// TIA Portal V17 export
// export: Created 2022-07-20T06:59:46.8680276Z, ExportSetting WithDefaults, DisplayName Totally Integrated Automation Portal, DisplayVersion V17, DisplayName TIA Portal Openness, DisplayVersion V17, DisplayName TIA Portal Version Control Interface, DisplayVersion V17, DisplayName SINAMICS Startdrive Advanced, DisplayVersion V17, DisplayName SINAMICS Startdrive G130, G150, S120, S150, SINAMICS MV, S210, DisplayVersion V17, DisplayName SINAMICS Startdrive G110M, G120, G120C, G120D, G120P, G115D, DisplayVersion V17, DisplayName STEP 7 Professional, DisplayVersion V17, DisplayName STEP 7 Safety, DisplayVersion V17, DisplayName WinCC Advanced, DisplayVersion V17
FUNCTION_BLOCK "FB10100_ModbusRtuManager"   // FB10100, LAD
TITLE = FB10100_ModbusRtuManager
{ S7_Optimized_Access := 'FALSE' }
AUTHOR : Jonathan
FAMILY : 1010x_MODBUS
VERSION : 1.0
// Release note : 
// 1.0 - Feature developped
// 
// Todo : 
// Générer une erreur si la communication reste en busy trop longtemps
// stored: AutoNumber false, IsIECCheckEnabled false, SetENOAutomatically false, UDAEnableTagReadback false
   VAR_INPUT
      InitialCall : Bool;
      ModbusPort : HW_ANY;
      ModbusBaudRate : UDInt;
      ModbusParity : UInt;
      StartCommunication : Bool;
      Reset : Bool;
      Max_ModbusSlaves : Int := 1;
   END_VAR
   VAR_OUTPUT
      Init_Done : Bool;
      Init_Error : Bool;
      Init_Status : Word;
      Comm_Done : Bool;
      Comm_Busy : Bool;
      Comm_Error : Bool;
      Comm_Status : Word;
   END_VAR
   VAR_IN_OUT
      CurrentSlaveNumber : Int;
      SlavesParameters : Array[1.."MAX_MODBUS_SLAVES"] of "stModbusRtuSlaveParameters";
      SlavesRequests : Array[1.."MAX_MODBUS_SLAVES"] of "stModbusRtuSlaveRequests";
      SlavesStates : Array[1.."MAX_MODBUS_SLAVES"] of "stModbusRtuSlaveStates";
   END_VAR
   VAR
      Modbus_Master_DB { ExternalAccessible := 'False'; ExternalVisible := 'False'; ExternalWritable := 'False'; S7_SetPoint := 'True'} : Modbus_Master;
      Modbus_Comm_Load_DB { S7_SetPoint := 'True'} : Modbus_Comm_Load;
   END_VAR
   VAR DB_SPECIFIC
      InitalisationDoneStored : Bool;
      LocalProcessStep : USInt;
      LocalCommRequest : Bool;
      LocalMode : USInt;
      LocalSlaveDataTemp { ExternalAccessible := 'False'; ExternalVisible := 'False'; ExternalWritable := 'False'; S7_SetPoint := 'True'} : "stModbusRtuDataPtr";
      LocalSlaveAdress : UInt;
      LocalSlaveDataAdress : UInt;
      Data_modbus_Dint { ExternalAccessible := 'False'; ExternalVisible := 'False'; ExternalWritable := 'False'} : DInt;
      Modbus_value_Number { ExternalAccessible := 'False'; ExternalVisible := 'False'; ExternalWritable := 'False'} : DInt;
      LocalSlaveDataLength : UInt;
      Data_modbus_Int : Int;
      TON_TimeOutNotDone { S7_SetPoint := 'True'} : TON_TIME;
      LocalSlaveCurrentNumber : Int;
   END_VAR
   VAR_TEMP
      LowWeight : Int;
      LowWeight_1 : Real;
      Highweight : Real;
   END_VAR
   // Modbus_Comm_Load_DB.STOP_BITS := 2;
BEGIN

REGION Network 1: Initilisation of the mode (4 = Half Duplex) / Put 4 value for Half Duplex mode
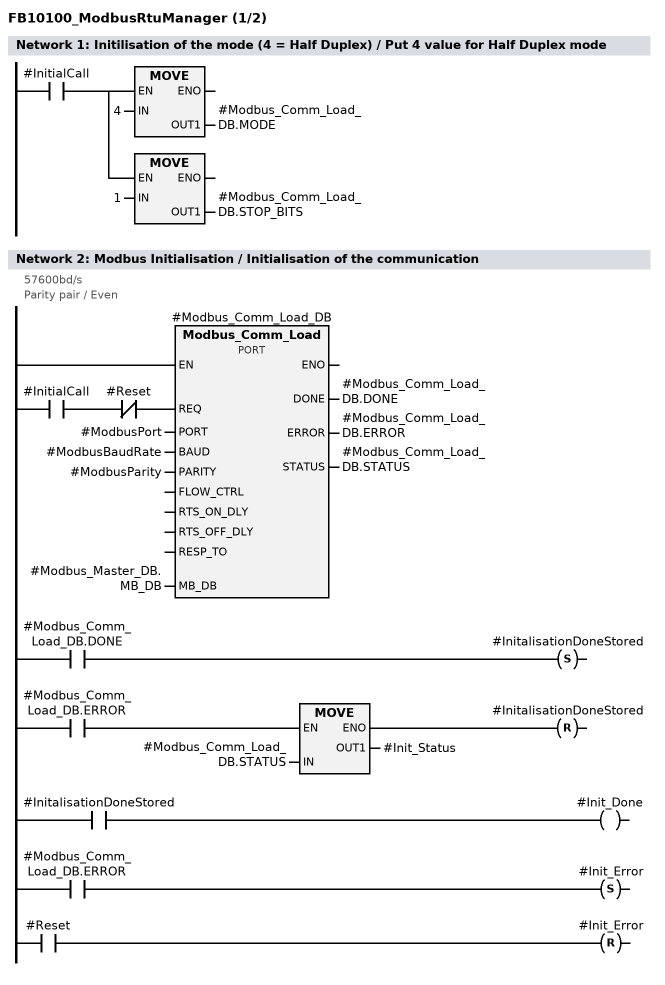
   RUNG wire#powerrail
      Contact( #InitialCall )
      wire#w1
      { S7_GenerateENO := "TRUE" } Move(in := 4, out1 => #Modbus_Comm_Load_DB.MODE)
   END_RUNG
   RUNG wire#w1
      { S7_GenerateENO := "TRUE" } Move(in := 1, out1 => #Modbus_Comm_Load_DB.STOP_BITS)
   END_RUNG
   // the same network as SCL:
   IF #InitialCall THEN
       #Modbus_Comm_Load_DB.MODE := 4;
       #Modbus_Comm_Load_DB.STOP_BITS := 1;
   END_IF;
END_REGION

REGION Network 2: Modbus Initialisation / Initialisation of the communication
   // 57600bd/s
   // Parity pair / Even
   RUNG wire#powerrail
      { S7_Templates := "[card := 0, port_type := PORT, word_type := UInt, dint_type := UDInt, mbbase_type := P2P_MB_BASE]" } #Modbus_Comm_Load_DB.Modbus_Comm_Load(REQ := wire#w1, PORT := #ModbusPort, BAUD := #ModbusBaudRate, PARITY := #ModbusParity, FLOW_CTRL :=, RTS_ON_DLY :=, RTS_OFF_DLY :=, RESP_TO :=, MB_DB := #Modbus_Master_DB.MB_DB, DONE => #Modbus_Comm_Load_DB.DONE, ERROR => #Modbus_Comm_Load_DB.ERROR, STATUS => #Modbus_Comm_Load_DB.STATUS)
   END_RUNG
   RUNG wire#powerrail
      Contact( #InitialCall )
      I_Contact( #Reset )
   END_RUNG wire#w1
   RUNG wire#powerrail
      Contact( #Modbus_Comm_Load_DB.DONE )
      S_Coil( #InitalisationDoneStored )
   END_RUNG
   RUNG wire#powerrail
      Contact( #Modbus_Comm_Load_DB.ERROR )
      { S7_GenerateENO := "TRUE" } Move(in := #Modbus_Comm_Load_DB.STATUS, out1 => #Init_Status)
      R_Coil( #InitalisationDoneStored )
   END_RUNG
   RUNG wire#powerrail
      Contact( #InitalisationDoneStored )
      Coil( #Init_Done )
   END_RUNG
   RUNG wire#powerrail
      Contact( #Modbus_Comm_Load_DB.ERROR )
      S_Coil( #Init_Error )
   END_RUNG
   RUNG wire#powerrail
      Contact( #Reset )
      R_Coil( #Init_Error )
   END_RUNG
   // the same network as SCL:
   // ENO of a box is taken as its EN; it also drops when the box reports an error
   #Modbus_Comm_Load_DB(REQ := #InitialCall AND NOT #Reset,   // Modbus_Comm_Load
                        PORT := #ModbusPort,
                        BAUD := #ModbusBaudRate,
                        PARITY := #ModbusParity,
                        MB_DB := #Modbus_Master_DB.MB_DB,
                        DONE => #Modbus_Comm_Load_DB.DONE,
                        ERROR => #Modbus_Comm_Load_DB.ERROR,
                        STATUS => #Modbus_Comm_Load_DB.STATUS);
   IF #Modbus_Comm_Load_DB.DONE THEN #InitalisationDoneStored := TRUE; END_IF;
   IF #Modbus_Comm_Load_DB.ERROR THEN
       #Init_Status := #Modbus_Comm_Load_DB.STATUS;
       #InitalisationDoneStored := FALSE;
   END_IF;
   #Init_Done := #InitalisationDoneStored;
   IF #Modbus_Comm_Load_DB.ERROR THEN #Init_Error := TRUE; END_IF;
   IF #Reset THEN #Init_Error := FALSE; END_IF;
END_REGION

REGION Network 3: Modbus Master Call / Master Exchange block
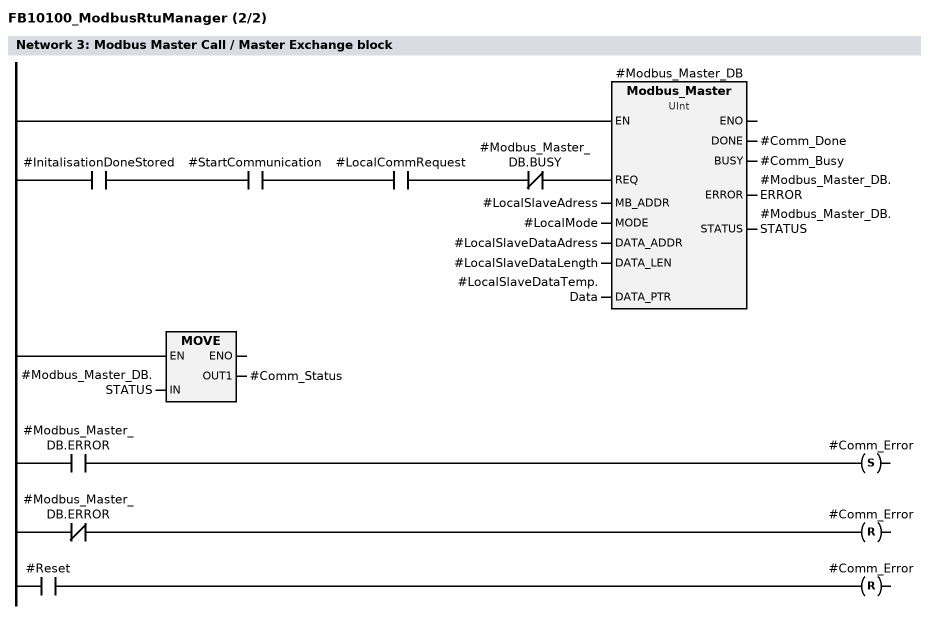
   RUNG wire#powerrail
      { S7_Templates := "[card := 0, word_type := UInt, dword_type := UDInt, byte_type := USInt, any_type := Variant]" } #Modbus_Master_DB.Modbus_Master(REQ := wire#w1, MB_ADDR := #LocalSlaveAdress, MODE := #LocalMode, DATA_ADDR := #LocalSlaveDataAdress, DATA_LEN := #LocalSlaveDataLength, DATA_PTR := #LocalSlaveDataTemp.Data, DONE => #Comm_Done, BUSY => #Comm_Busy, ERROR => #Modbus_Master_DB.ERROR, STATUS => #Modbus_Master_DB.STATUS)
   END_RUNG
   RUNG wire#powerrail
      Contact( #InitalisationDoneStored )
      Contact( #StartCommunication )
      Contact( #LocalCommRequest )
      I_Contact( #Modbus_Master_DB.BUSY )
   END_RUNG wire#w1
   RUNG wire#powerrail
      { S7_GenerateENO := "TRUE" } Move(in := #Modbus_Master_DB.STATUS, out1 => #Comm_Status)
   END_RUNG
   RUNG wire#powerrail
      Contact( #Modbus_Master_DB.ERROR )
      S_Coil( #Comm_Error )
   END_RUNG
   RUNG wire#powerrail
      I_Contact( #Modbus_Master_DB.ERROR )
      R_Coil( #Comm_Error )
   END_RUNG
   RUNG wire#powerrail
      Contact( #Reset )
      R_Coil( #Comm_Error )
   END_RUNG
   // the same network as SCL:
   #Modbus_Master_DB(REQ := #InitalisationDoneStored AND #StartCommunication AND #LocalCommRequest AND NOT #Modbus_Master_DB.BUSY,   // Modbus_Master
                     MB_ADDR := #LocalSlaveAdress,
                     MODE := #LocalMode,
                     DATA_ADDR := #LocalSlaveDataAdress,
                     DATA_LEN := #LocalSlaveDataLength,
                     DATA_PTR := #LocalSlaveDataTemp.Data,
                     DONE => #Comm_Done,
                     BUSY => #Comm_Busy,
                     ERROR => #Modbus_Master_DB.ERROR,
                     STATUS => #Modbus_Master_DB.STATUS);
   #Comm_Status := #Modbus_Master_DB.STATUS;
   IF #Modbus_Master_DB.ERROR THEN #Comm_Error := TRUE; END_IF;
   IF NOT #Modbus_Master_DB.ERROR THEN #Comm_Error := FALSE; END_IF;
   IF #Reset THEN #Comm_Error := FALSE; END_IF;
END_REGION

REGION Network 4 (SCL): Step 0 : Wait for start Modbus Communication / Step 0 : Start Modbus communication
   #CurrentSlaveNumber := #LocalSlaveCurrentNumber;

   IF #Comm_Error OR NOT #StartCommunication THEN
       #LocalProcessStep := 0;
       #LocalCommRequest := FALSE;
   ELSE
       IF #LocalProcessStep = 0 THEN
           IF #StartCommunication THEN
               IF #LocalSlaveCurrentNumber <= 0 OR #LocalSlaveCurrentNumber > #Max_ModbusSlaves THEN
                   #LocalSlaveCurrentNumber := 1;
               END_IF;
               #LocalProcessStep := 1;
           END_IF;
       END_IF;
   END_IF;
END_REGION

REGION Network 5 (SCL): Step 1 : Find the Next Modbus Slave to refresh in read or write mode / Step 1 :
   IF #LocalProcessStep = 1 THEN
       IF #LocalSlaveCurrentNumber <= 0 OR #LocalSlaveCurrentNumber > #Max_ModbusSlaves THEN
           #LocalProcessStep := 0;
       ELSE
           #SlavesStates[#LocalSlaveCurrentNumber].UpdateDone := FALSE;
           IF #SlavesRequests[#LocalSlaveCurrentNumber].StartRequest THEN
               #LocalCommRequest := #SlavesRequests[#LocalSlaveCurrentNumber].StartRequest;
               #LocalSlaveAdress := #SlavesParameters[#LocalSlaveCurrentNumber].SlaveAddress;
               #LocalSlaveDataAdress := #SlavesParameters[#LocalSlaveCurrentNumber].DataAddress;
               #LocalSlaveDataLength := #SlavesParameters[#LocalSlaveCurrentNumber].DataLength;
               #LocalMode := #SlavesParameters[#LocalSlaveCurrentNumber].Mode;
               #LocalSlaveDataTemp := #SlavesStates[#LocalSlaveCurrentNumber].DataToSend;
               #LocalProcessStep := 5;
           ELSE
               #LocalSlaveCurrentNumber := #LocalSlaveCurrentNumber + 1;
               #LocalProcessStep := 1;
           END_IF; 

       END_IF; 
   END_IF;
END_REGION

REGION Network 6 (SCL): Step 5 : Wait for update done and go to Step 1 with next Slave adress / Step 5 : Wait done
   #TON_TimeOutNotDone(IN := #LocalProcessStep = 5 AND NOT(#Comm_Done) AND #Comm_Busy,
                       PT := T#10s);

   IF #LocalProcessStep = 5 THEN
       IF #Comm_Done OR #TON_TimeOutNotDone.Q THEN
           IF #SlavesParameters[#LocalSlaveCurrentNumber].Mode = 0 THEN
               #SlavesStates[#LocalSlaveCurrentNumber].DataToReceive.Data := #LocalSlaveDataTemp.Data;
           END_IF;

           #SlavesStates[#LocalSlaveCurrentNumber].UpdateDone := TRUE;
           #LocalSlaveCurrentNumber := #LocalSlaveCurrentNumber + 1;
           #LocalProcessStep := 1;
       ELSIF #TON_TimeOutNotDone.Q THEN
           #LocalCommRequest := FALSE;
           #LocalSlaveCurrentNumber := #LocalSlaveCurrentNumber + 1;
           #LocalProcessStep := 1;
       END_IF;
   END_IF;
END_REGION
END_FUNCTION_BLOCK
